(* PLC project CoDeSys External Library Template, WAGO e!COCKPIT e!COCKPIT, author 3S - Smart Software Solutions GmbH *)
(* stored: creationDateTime 2019-10-29T12:37:19.3050686, version 3.5.5.30, modificationDateTime 2019-10-29T12:36:39.3744516, organization 3S - Smart Software Solutions GmbH *)
(* Library project template with all possible element types, docu and a sample project structure *)

(* values of enumModbusStatus: BrakKomunikacji: problem z komunikacją; KomunikacjaPrawidlowa: komunikacja przebiegła prawidłowo *)

(* Nazwa bloku: Enumeracja - definicja kodów błędów w komunikacji modbus Projekt: Bałtyckie Centrum Biznesu Budynek 2 Firma: Solwena Autor: Marcin Szumiło Wersja: 0.1.0.1 - 2017-01-10 *)
{attribute 'qualified_only'}
{attribute 'strict'}
TYPE enumModbusStatus : (BrakKomunikacji := 1, KomunikacjaPrawidlowa := 2);
END_TYPE
